{attribute 'GeneratedUsingTerminal: AT2041-0250-0019'}
{attribute addProperty BoxType "AT2041-0250-0019"}
{attribute addProperty Id "A_0103_AT2042_5250_0018_AT2042_5250AT2042_01D6DEDF80"}
{attribute addProperty CRC "1641063610"}
{attribute addProperty Size "80"}
TYPE A_0041_AT2041_0250_0019_61D0A4BA EXTENDS AT2041_86175B41 :
STRUCT
	{attribute addProperty Name "A_0103_AT2042_5250_0018_AT2042_5250"}
	{attribute addProperty PreviousPort "A_0041(AT2041-0250-0019) : B"}
	A_0103_AT2042_5250_0018_AT2042_5250 : AT2042_01D6DEDF;
END_STRUCT
END_TYPE

(* stored: Version 1.2.0.0, ProductVersion 3.1.4024.9
   DUT A_0041_AT2041_0250_0019_61D0A4BA: Id {6051da36-e164-46bc-97e1-5d13147a14c0} *)
